TYPE OPC_UA_BOOL :
STRUCT
	NodeID				: ST_UANodeID;
	NodeHdl				: DWORD;
	SizeOfDataType		: UDINT;
	NodeAddInfo			: ST_UANodeAdditionalInfo;
	TargetVar			: POINTER TO BOOL;
END_STRUCT
END_TYPE

(* stored: Version 1.1.0.1, ProductVersion 3.1.4024.9
   DUT OPC_UA_BOOL: Id {7afe51be-c3ee-456b-807a-9d10ca5c8d1b} *)
